// TIA Portal V16 export
// export: Created 2022-07-21T09:35:31.1306103Z, ExportSetting WithDefaults, DisplayName Totally Integrated Automation Portal, DisplayVersion V16 Update 4, DisplayName TIA Portal Version Control Interface, DisplayVersion V16 Update 2, DisplayName TIA Portal Openness, DisplayVersion V16 Update 4, DisplayName SINAMICS Startdrive Advanced, DisplayVersion V16 Update 5, DisplayName SINAMICS Startdrive G130, G150, S120, S150, SINAMICS MV, S210, DisplayVersion V16 Update 5, DisplayName SINAMICS Startdrive G110M, G120, G120C, G120D, G120P, G115D, DisplayVersion V16 Update 5, DisplayName STEP 7 Professional, DisplayVersion V16 Update 4, DisplayName STEP 7 Safety, DisplayVersion V16, DisplayName WinCC Advanced, DisplayVersion V16 Update 4
FUNCTION_BLOCK "fbSignal"   // FB37, LAD
TITLE = Signal handling / Obsługa sygnału
{ S7_Optimized_Access := 'TRUE' }
VERSION : 0.1
// stored: AutoNumber true, IsIECCheckEnabled false, IsRetainMemResEnabled false, MemoryReserve 100, SetENOAutomatically false, UDAEnableTagReadback false
   VAR_INPUT
      inSignal : Bool;   // Sygnał wejściowy / Input signal
      inNC : Bool;   // NC = true, NO = false
   END_VAR
   VAR_OUTPUT
      ouSignal : "typeSignal";   // Sygnał wyjściowy - okupacja, zbocze narastające i opadające / Output signal - occupation, rising & falling edge
   END_VAR
   VAR
      sPosEdgeMem : Bool;
      sNegEdgeMem : Bool;
   END_VAR
   VAR_TEMP
      tSignal : Bool;
   END_VAR
BEGIN

REGION Network 1: Signal handling / Obsługa sygnału
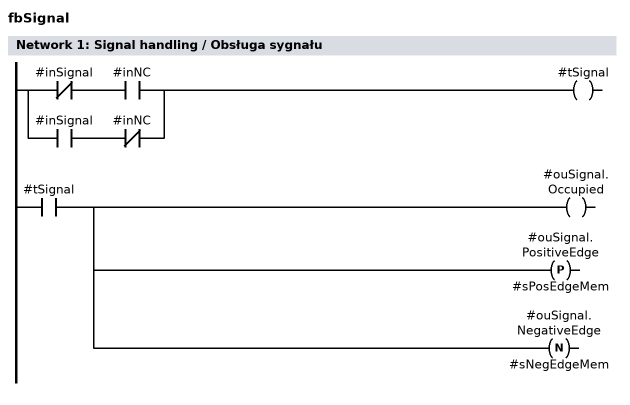
   #tSignal := (NOT #inSignal AND #inNC) OR (#inSignal AND NOT #inNC);
   #ouSignal.Occupied := #tSignal;
   #ouSignal.PositiveEdge := #tSignal AND NOT #sPosEdgeMem;   // rising edge
   #sPosEdgeMem := #tSignal;
   #ouSignal.NegativeEdge := NOT #tSignal AND #sNegEdgeMem;   // falling edge
   #sNegEdgeMem := #tSignal;
END_REGION
END_FUNCTION_BLOCK
